{attribute 'GeneratedUsingTerminal: EK1100-0000-0018'}
{attribute addProperty BoxType "EK1100-0000-0018"}
{attribute addProperty Id "Beckhoff_EQ3xxxEK1122Beckhoff_EQ3xxxEK1122_A1C56A21718"}
{attribute addProperty CRC "2837491862"}
{attribute addProperty Size "718"}
{attribute addProperty Name "Beckhoff EQ3xxx"}
TYPE Beckhoff_EQ3xxx_A920B096 EXTENDS EK1100_1FC0878B :
STRUCT
	{attribute addProperty Name "Beckhoff EQ3xxxEK1122"}
	{attribute addProperty PreviousPort "Beckhoff EQ3xxx : B"}
	Beckhoff_EQ3xxxEK1122 : Beckhoff_EQ3xxxEK1122_A1C56A21;
END_STRUCT
END_TYPE

(* stored: Version 1.2.0.0, ProductVersion 3.1.4024.11
   DUT Beckhoff_EQ3xxx_A920B096: Id {94d17cd8-b2ef-488e-8cc7-e4b91a304566} *)
